// TIA Portal V19 export
DATA_BLOCK "CTrk"   // DB43
// stored: MemoryReserve 100
   VAR RETAIN
      Last_C_ID : DInt;   // Ultimo ID assegnato
      Empty : "CTrk_Item";   // Item ausiliario per cancellazione dati
      A01_Preparation : "CTrk_Item";   // Prossimo materiale su Coil in prepazione = Su aspo fuori linea
      A01_Processing : "CTrk_Item";   // Materiale in lavoro su Area 01
      A02_Next : "CTrk_Item";   // Prossimo materiale in arrivo per esecuzione dei SG
      A02_Processing : "CTrk_Item";   // Materiale su stampo in esecuzione SG
      A02_Consumed : "CTrk_Item";   // Materiale uscita completamente dal taglio
   END_VAR
BEGIN
END_DATA_BLOCK
